(*
    This function block reports the results from the tests using the built-in ADSLOGSTR functionality
    provided by the Tc2_System library. This sends the result using ADS, which is consumed by the error list
    of Visual Studio.
*)
FUNCTION_BLOCK FB_ADSTestResultFormatter IMPLEMENTS I_TestResultFormatter
VAR
    (* Although we can print a message no #1 prior to message no #2, the message #2 can still be displayed before
       message #1, most likely because of some delay of the ADS data. To workaround this, we add a small delay between
       transmission of the ADS messages. *)
    ADSDelayTimer : Tc2_Standard.TON := (PT := T#300MS);
    LastPrintState : USINT := 0;
    PrintState : USINT := 0;
END_VAR

METHOD Format
VAR_INPUT
    (* The total amount of test suites *)
    AmountOfTestSuites    : UINT;
    (* The total amount of test cases (for all test function blocks) *)
    AmountOfTestCases    : UINT;
    (* The total amount of test cases that had all ASSERTS successful *)
    AmountOfSuccessfulTestCases    : UINT;
    (* The total amount of test cases that had at least one ASSERT failed *)
    AmountOfFailedTestCases    : UINT;
END_VAR
VAR_OUTPUT
    Busy : BOOL;
END_VAR
VAR
    ErrorCode : DINT;
END_VAR
CASE PrintState OF
    0 :
        LastPrintState := PrintState;
        PrintState := 100;
        Busy := TRUE;
    1 :
        GVL_TcUnit.AdsLogger.WriteLog(MsgFmtStr := '%s',
                                      StrArg := '| ==========TESTS FINISHED RUNNING==========');
        LastPrintState := PrintState;
        PrintState := 100;
        Busy := TRUE;
    2 :
        GVL_TcUnit.AdsLogger.WriteLog(MsgFmtStr := '| Test suites: %s',
                                      StrArg := UINT_TO_STRING(AmountOfTestSuites));
        LastPrintState := PrintState;
        PrintState := 100;
        Busy := TRUE;
    3 :
        GVL_TcUnit.AdsLogger.WriteLog(MsgFmtStr := '| Tests: %s',
                                      StrArg := UINT_TO_STRING(AmountOfTestCases));
        LastPrintState := PrintState;
        PrintState := 100;
        Busy := TRUE;
    4 :
        GVL_TcUnit.AdsLogger.WriteLog(MsgFmtStr := '| Successful tests: %s',
                                      StrArg := UINT_TO_STRING(AmountOfSuccessfulTestCases));
        LastPrintState := PrintState;
        PrintState := 100;
        Busy := TRUE;
    5 :
        GVL_TcUnit.AdsLogger.WriteLog(MsgFmtStr := '| Failed tests: %s',
                                      StrArg := UINT_TO_STRING(AmountOfFailedTestCases));
        LastPrintState := PrintState;
        PrintState := 100;
        Busy := TRUE;
    6 :
        GVL_TcUnit.AdsLogger.WriteLog(MsgFmtStr := '%s',
                                      StrArg := '| ======================================');
        LastPrintState := PrintState;
        PrintState := 100;
        Busy := TRUE;
    7 :
        Busy := FALSE;
    100 :
        ADSDelayTimer(IN := TRUE);
        IF ADSDelayTimer.Q THEN
            ADSDelayTimer(IN := FALSE);
            PrintState := LastPrintState + 1;
        END_IF
        Busy := TRUE;
END_CASE
END_METHOD

END_FUNCTION_BLOCK

(* stored: Version 1.1.0.1, ProductVersion 3.1.4022.18
   POU FB_ADSTestResultFormatter: Id {d14d6247-3ce3-459f-be22-6ee3520279ed}, SpecialFunc None
   Method Format: Id {dba8c729-8b99-4be3-97cd-3a4fea4cd051} *)
